// TIA Portal project "SemaforV1" (V15.1)

(* hardware
DEVICE "S71500/ET200MP station_1"  S7-1500 station
   slot 0: "Rail_0"  Rack  6ES7 590-1***0-0AA0
   slot 1: "PLC_1"  CPU 1513-1 PN  6ES7 513-1AL02-0AB0  V2.6
      slot 3: "CPU display_1"  6ES7591-1AA00-0AA0
DEVICE "HMI_1"  KTP900 Basic PN
   slot 0: "HMI_1"  KTP900 Basic PN  6AV2 123-2JB03-0AX0  15.1.0.0
   slot 1: "HMI_RT_1"  KTP900 Basic PN  6AV2 123-2JB03-0AX0  15.1.0.0
   slot 5: "HMI_1.IE_CP_1"  PROFINET Interface  15.0.1.0
      slot 1: "PROFINET Interface_1"  PROFINET Interface
         slot 1: "Port_1"  Port
*)

// ===== PLC "PLC_1"  CPU 1513-1 PN =====

VAR_GLOBAL   // PLC tag table "Default tag table"
   "Clock_Byte" AT %MB0 : Byte;
   "Clock_10Hz" AT %M0.0 : Bool;
   "Clock_5Hz" AT %M0.1 : Bool;
   "Clock_2.5Hz" AT %M0.2 : Bool;
   "Clock_2Hz" AT %M0.3 : Bool;
   "Clock_1.25Hz" AT %M0.4 : Bool;
   "Clock_1Hz" AT %M0.5 : Bool;
   "Clock_0.625Hz" AT %M0.6 : Bool;
   "Clock_0.5Hz" AT %M0.7 : Bool;
END_VAR

DATA_BLOCK "Semafor_1_variabile"   // DB1
{ S7_Optimized_Access := 'TRUE' }
VERSION : 0.1
   VAR
      "mod functionare" : UInt;
      timp_verde : Time;
      timp_galben : Time;
      timp_rosu : Time;
      verde_on : Bool;
      galben_on : Bool;
      rosu_on : Bool;
      galben_intermitent : Bool;
   END_VAR
BEGIN
END_DATA_BLOCK

DATA_BLOCK "Semafor_2_variabile"   // DB2
{ S7_Optimized_Access := 'TRUE' }
VERSION : 0.1
   VAR
      "mod functionare" : UInt;
      timp_verde : Time;
      timp_galben : Time;
      timp_rosu : Time;
      verde_on : Bool;
      galben_on : Bool;
      rosu_on : Bool;
      galben_intermitent : Bool;
   END_VAR
BEGIN
END_DATA_BLOCK

DATA_BLOCK "Semafor_3_variabile"   // DB3
{ S7_Optimized_Access := 'TRUE' }
VERSION : 0.1
   VAR
      "mod functionare" : UInt;
      timp_verde : Time;
      timp_galben : Time;
      timp_rosu : Time;
      verde_on : Bool;
      galben_on : Bool;
      rosu_on : Bool;
      galben_intermitent : Bool;
   END_VAR
BEGIN
END_DATA_BLOCK

DATA_BLOCK "Semafor2"   // DB4
{ S7_Optimized_Access := 'TRUE' }
VERSION : 0.1
// stored: InstanceOfName Semafor_fct
"Semafor_fct"
BEGIN
END_DATA_BLOCK

DATA_BLOCK "Semafor3"   // DB5
{ S7_Optimized_Access := 'TRUE' }
VERSION : 0.1
// stored: InstanceOfName Semafor_fct
"Semafor_fct"
BEGIN
END_DATA_BLOCK

DATA_BLOCK "Semafor1"   // DB6
{ S7_Optimized_Access := 'TRUE' }
VERSION : 0.1
// stored: InstanceOfName Semafor_fct
"Semafor_fct"
BEGIN
END_DATA_BLOCK

DATA_BLOCK "Semafor_4_variabile"   // DB7
{ S7_Optimized_Access := 'TRUE' }
VERSION : 0.1
   VAR
      "mod functionare" : UInt;
      timp_verde : Time;
      timp_galben : Time;
      timp_rosu : Time;
      verde_on : Bool;
      galben_on : Bool;
      rosu_on : Bool;
      galben_intermitent : Bool;
   END_VAR
BEGIN
END_DATA_BLOCK

DATA_BLOCK "Semafor4"   // DB8
{ S7_Optimized_Access := 'TRUE' }
VERSION : 0.1
// stored: InstanceOfName Semafor_fct
"Semafor_fct"
BEGIN
END_DATA_BLOCK

FUNCTION_BLOCK "Semafor_fct"   // FB1, LAD
{ S7_Optimized_Access := 'TRUE' }
VERSION : 0.1
   VAR_INPUT
      timp_verde : Time;
      timp_galben : Time;
      timp_rosu : Time;
   END_VAR
   VAR_OUTPUT
      verde_on : Bool;
      galben_on : Bool;
      rosu_on : Bool;
      galben_intermitnet : Bool;
   END_VAR
   VAR_IN_OUT
      mod_functionare : UInt;
   END_VAR
   VAR
      pornire_normal : Bool;
      reseteaza_bucla : Bool;
      porneste_verde : Bool;
      porneste_galben : Bool;
      porneste_rosu : Bool;
      timer_verde : TON_TIME;
      timer_galben : TON_TIME;
      timer_rosu : TON_TIME;
      rising_edge : Bool;
      testing : Bool;
      timp_verde_secunde : Time;
      timp_rosu_secunde : Time;
      timp_galben_secunde : Time;
   END_VAR
   VAR_TEMP   // added for the SCL form of the ladder/FBD networks
      _w1 : Bool;
   END_VAR
BEGIN

REGION Network 1: timp in secunde
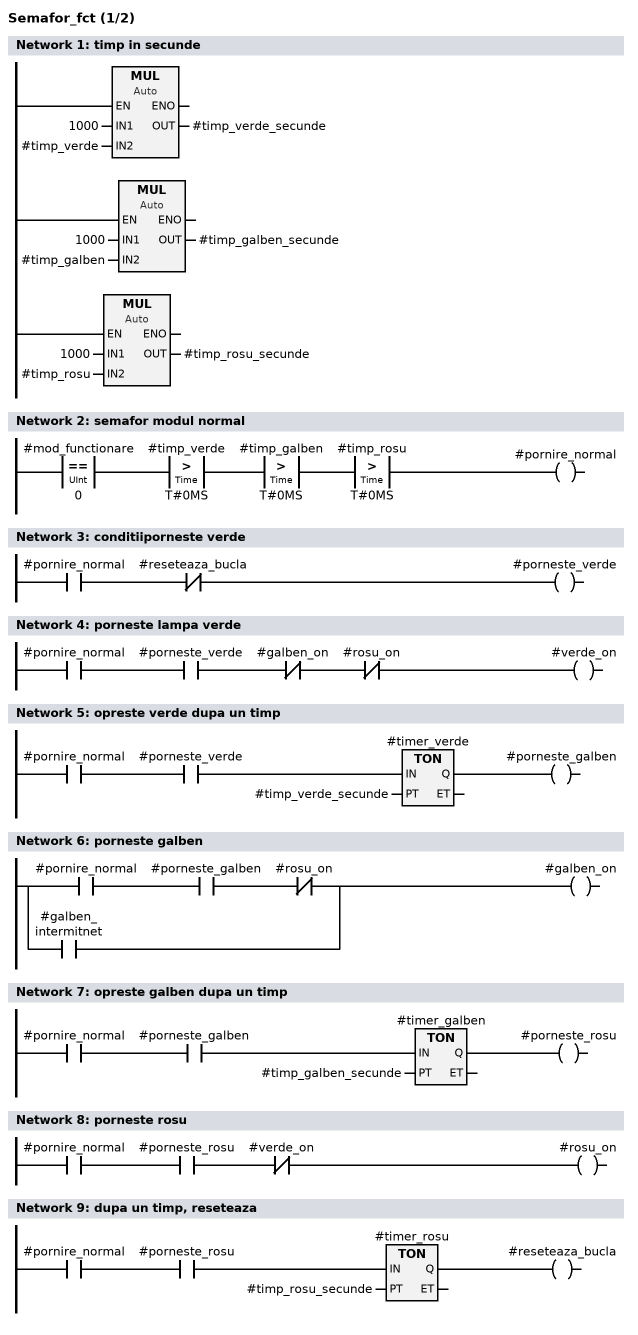
   RUNG wire#powerrail
      Mul(in1 := 1000, in2 := #timp_verde, out => #timp_verde_secunde)
   END_RUNG
   RUNG wire#powerrail
      Mul(in1 := 1000, in2 := #timp_galben, out => #timp_galben_secunde)
   END_RUNG
   RUNG wire#powerrail
      Mul(in1 := 1000, in2 := #timp_rosu, out => #timp_rosu_secunde)
   END_RUNG
   // the same network as SCL:
   #timp_verde_secunde := 1000 * #timp_verde;
   #timp_galben_secunde := 1000 * #timp_galben;
   #timp_rosu_secunde := 1000 * #timp_rosu;
END_REGION

REGION Network 2: semafor modul normal
   RUNG wire#powerrail
      { S7_Templates := "SrcType := UInt" } EQ_Contact(in1 := #mod_functionare, in2 := 0)
      { S7_Templates := "SrcType := Time" } GT_Contact(in1 := #timp_verde, in2 := T#0MS)
      { S7_Templates := "SrcType := Time" } GT_Contact(in1 := #timp_galben, in2 := T#0MS)
      { S7_Templates := "SrcType := Time" } GT_Contact(in1 := #timp_rosu, in2 := T#0MS)
      Coil( #pornire_normal )
   END_RUNG
   // the same network as SCL:
   #pornire_normal := (#mod_functionare = 0) AND (#timp_verde > T#0MS) AND (#timp_galben > T#0MS) AND (#timp_rosu > T#0MS);
END_REGION

REGION Network 3: conditiiporneste verde
   RUNG wire#powerrail
      Contact( #pornire_normal )
      I_Contact( #reseteaza_bucla )
      Coil( #porneste_verde )
   END_RUNG
   // the same network as SCL:
   #porneste_verde := #pornire_normal AND NOT #reseteaza_bucla;
END_REGION

REGION Network 4: porneste lampa verde
   RUNG wire#powerrail
      Contact( #pornire_normal )
      Contact( #porneste_verde )
      I_Contact( #galben_on )
      I_Contact( #rosu_on )
      Coil( #verde_on )
   END_RUNG
   // the same network as SCL:
   #verde_on := #pornire_normal AND #porneste_verde AND NOT #galben_on AND NOT #rosu_on;
END_REGION

REGION Network 5: opreste verde dupa un timp
   #timer_verde(IN := #pornire_normal AND #porneste_verde, PT := #timp_verde_secunde);   // TON
   #porneste_galben := #timer_verde.Q;
END_REGION

REGION Network 6: porneste galben
   RUNG wire#powerrail
      Contact( #pornire_normal )
      Contact( #porneste_galben )
      I_Contact( #rosu_on )
      wire#w1
      Coil( #galben_on )
   END_RUNG
   RUNG wire#powerrail
      Contact( #galben_intermitnet )
   END_RUNG wire#w1
   // the same network as SCL:
   #galben_on := (#pornire_normal AND #porneste_galben AND NOT #rosu_on) OR #galben_intermitnet;
END_REGION

REGION Network 7: opreste galben dupa un timp
   #timer_galben(IN := #pornire_normal AND #porneste_galben, PT := #timp_galben_secunde);   // TON
   #porneste_rosu := #timer_galben.Q;
END_REGION

REGION Network 8: porneste rosu
   RUNG wire#powerrail
      Contact( #pornire_normal )
      Contact( #porneste_rosu )
      I_Contact( #verde_on )
      Coil( #rosu_on )
   END_RUNG
   // the same network as SCL:
   #rosu_on := #pornire_normal AND #porneste_rosu AND NOT #verde_on;
END_REGION

REGION Network 9: dupa un timp, reseteaza
   #timer_rosu(IN := #pornire_normal AND #porneste_rosu, PT := #timp_rosu_secunde);   // TON
   #reseteaza_bucla := #timer_rosu.Q;
END_REGION

REGION Network 10: toggle rising edge pt SR la galben intermitent pe avarie
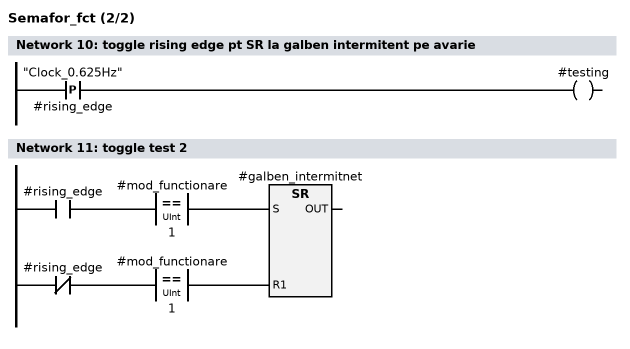
   RUNG wire#powerrail
      P_Contact(operand := "Clock_0.625Hz", bit := #rising_edge)
      Coil( #testing )
   END_RUNG
   // the same network as SCL:
   #_w1 := "Clock_0.625Hz" AND NOT #rising_edge;   // rising edge of "Clock_0.625Hz"
   #rising_edge := "Clock_0.625Hz";
   #testing := #_w1;
END_REGION

REGION Network 11: toggle test 2
   RUNG wire#powerrail
      Contact( #rising_edge )
      { S7_Templates := "SrcType := UInt" } EQ_Contact(in1 := #mod_functionare, in2 := 1)
      S_SR(operand := #galben_intermitnet, r1 := wire#w1)
   END_RUNG
   RUNG wire#powerrail
      I_Contact( #rising_edge )
      { S7_Templates := "SrcType := UInt" } EQ_Contact(in1 := #mod_functionare, in2 := 1)
   END_RUNG wire#w1
   // the same network as SCL:
   IF #rising_edge AND (#mod_functionare = 1) THEN
       #galben_intermitnet := TRUE;   // SR flip-flop
   END_IF;
   IF NOT #rising_edge AND (#mod_functionare = 1) THEN #galben_intermitnet := FALSE; END_IF;
END_REGION
END_FUNCTION_BLOCK

ORGANIZATION_BLOCK "Main"   // OB1, LAD, ProgramCycle
TITLE = "Main Program Sweep (Cycle)"
{ S7_Optimized_Access := 'TRUE' }
VERSION : 0.1
   VAR_INPUT
      Initial_Call : Bool;   // Initial call of this OB
      Remanence : Bool;   // =True, if remanent data are available
   END_VAR
   VAR_TEMP   // added for the SCL form of the ladder/FBD networks
      _w1 : Bool;
   END_VAR
BEGIN

REGION Network 1: porneste semafoarele 2 si 3 daca 1 si 4 sunt pe rosu
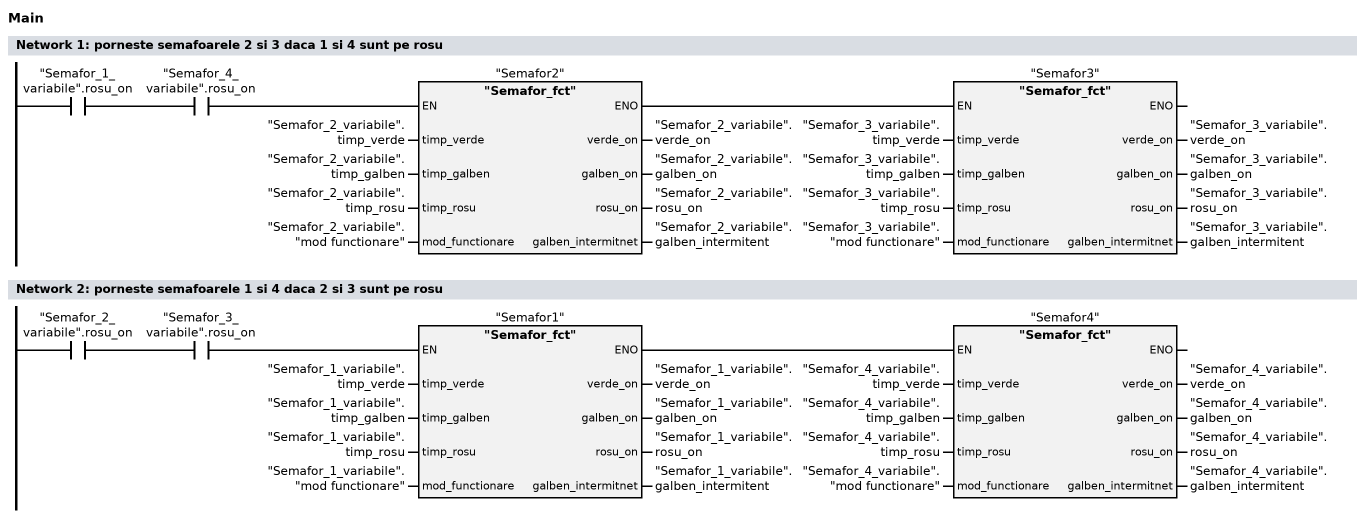
   RUNG wire#powerrail
      Contact( "Semafor_1_variabile".rosu_on )
      Contact( "Semafor_4_variabile".rosu_on )
      "Semafor2"(timp_verde := "Semafor_2_variabile".timp_verde, timp_galben := "Semafor_2_variabile".timp_galben, timp_rosu := "Semafor_2_variabile".timp_rosu, mod_functionare := "Semafor_2_variabile"."mod functionare", verde_on => "Semafor_2_variabile".verde_on, galben_on => "Semafor_2_variabile".galben_on, rosu_on => "Semafor_2_variabile".rosu_on, galben_intermitnet => "Semafor_2_variabile".galben_intermitent)
      "Semafor3"(timp_verde := "Semafor_3_variabile".timp_verde, timp_galben := "Semafor_3_variabile".timp_galben, timp_rosu := "Semafor_3_variabile".timp_rosu, mod_functionare := "Semafor_3_variabile"."mod functionare", verde_on => "Semafor_3_variabile".verde_on, galben_on => "Semafor_3_variabile".galben_on, rosu_on => "Semafor_3_variabile".rosu_on, galben_intermitnet => "Semafor_3_variabile".galben_intermitent)
   END_RUNG
   // the same network as SCL:
   "Semafor2"(EN := "Semafor_1_variabile".rosu_on AND "Semafor_4_variabile".rosu_on,   // "Semafor_fct"
              timp_verde := "Semafor_2_variabile".timp_verde,
              timp_galben := "Semafor_2_variabile".timp_galben,
              timp_rosu := "Semafor_2_variabile".timp_rosu,
              mod_functionare := "Semafor_2_variabile"."mod functionare",
              verde_on => "Semafor_2_variabile".verde_on,
              galben_on => "Semafor_2_variabile".galben_on,
              rosu_on => "Semafor_2_variabile".rosu_on,
              galben_intermitnet => "Semafor_2_variabile".galben_intermitent,
              ENO => #_w1);
   IF #_w1 THEN
       "Semafor3"(timp_verde := "Semafor_3_variabile".timp_verde,   // "Semafor_fct"
                  timp_galben := "Semafor_3_variabile".timp_galben,
                  timp_rosu := "Semafor_3_variabile".timp_rosu,
                  mod_functionare := "Semafor_3_variabile"."mod functionare",
                  verde_on => "Semafor_3_variabile".verde_on,
                  galben_on => "Semafor_3_variabile".galben_on,
                  rosu_on => "Semafor_3_variabile".rosu_on,
                  galben_intermitnet => "Semafor_3_variabile".galben_intermitent);
   END_IF;
END_REGION

REGION Network 2: porneste semafoarele 1 si 4 daca 2 si 3 sunt pe rosu
   RUNG wire#powerrail
      Contact( "Semafor_2_variabile".rosu_on )
      Contact( "Semafor_3_variabile".rosu_on )
      "Semafor1"(timp_verde := "Semafor_1_variabile".timp_verde, timp_galben := "Semafor_1_variabile".timp_galben, timp_rosu := "Semafor_1_variabile".timp_rosu, mod_functionare := "Semafor_1_variabile"."mod functionare", verde_on => "Semafor_1_variabile".verde_on, galben_on => "Semafor_1_variabile".galben_on, rosu_on => "Semafor_1_variabile".rosu_on, galben_intermitnet => "Semafor_1_variabile".galben_intermitent)
      "Semafor4"(timp_verde := "Semafor_4_variabile".timp_verde, timp_galben := "Semafor_4_variabile".timp_galben, timp_rosu := "Semafor_4_variabile".timp_rosu, mod_functionare := "Semafor_4_variabile"."mod functionare", verde_on => "Semafor_4_variabile".verde_on, galben_on => "Semafor_4_variabile".galben_on, rosu_on => "Semafor_4_variabile".rosu_on, galben_intermitnet => "Semafor_4_variabile".galben_intermitent)
   END_RUNG
   // the same network as SCL:
   "Semafor1"(EN := "Semafor_2_variabile".rosu_on AND "Semafor_3_variabile".rosu_on,   // "Semafor_fct"
              timp_verde := "Semafor_1_variabile".timp_verde,
              timp_galben := "Semafor_1_variabile".timp_galben,
              timp_rosu := "Semafor_1_variabile".timp_rosu,
              mod_functionare := "Semafor_1_variabile"."mod functionare",
              verde_on => "Semafor_1_variabile".verde_on,
              galben_on => "Semafor_1_variabile".galben_on,
              rosu_on => "Semafor_1_variabile".rosu_on,
              galben_intermitnet => "Semafor_1_variabile".galben_intermitent,
              ENO => #_w1);
   IF #_w1 THEN
       "Semafor4"(timp_verde := "Semafor_4_variabile".timp_verde,   // "Semafor_fct"
                  timp_galben := "Semafor_4_variabile".timp_galben,
                  timp_rosu := "Semafor_4_variabile".timp_rosu,
                  mod_functionare := "Semafor_4_variabile"."mod functionare",
                  verde_on => "Semafor_4_variabile".verde_on,
                  galben_on => "Semafor_4_variabile".galben_on,
                  rosu_on => "Semafor_4_variabile".rosu_on,
                  galben_intermitnet => "Semafor_4_variabile".galben_intermitent);
   END_IF;
END_REGION
END_ORGANIZATION_BLOCK

(* ===== HMI "HMI_RT_1" =====
system functions are stored by id; their names below are inferred from use
connection "HMI_Connection_1": ETHERNET, SMART_S7_1500_OMS

HMI tags "Default tag table"
   "Tag_ScreenNumber" : UInt, internal
   "Semafor_1_variabile_timp_verde" : Time = PLC Semafor_1_variabile.timp_verde, 1 s
   "Semafor_1_variabile_timp_galben" : Time = PLC Semafor_1_variabile.timp_galben, 1 s
   "Semafor_1_variabile_timp_rosu" : Time = PLC Semafor_1_variabile.timp_rosu, 1 s
   "Semafor_2_variabile_timp_verde" : Time = PLC Semafor_2_variabile.timp_verde, 1 s
   "Semafor_2_variabile_timp_galben" : Time = PLC Semafor_2_variabile.timp_galben, 1 s
   "Semafor_2_variabile_timp_rosu" : Time = PLC Semafor_2_variabile.timp_rosu, 1 s
   "Semafor_3_variabile_timp_galben" : Time = PLC Semafor_3_variabile.timp_galben, 1 s
   "Semafor_3_variabile_timp_rosu" : Time = PLC Semafor_3_variabile.timp_rosu, 1 s
   "Semafor_4_variabile_timp_verde" : Time = PLC Semafor_4_variabile.timp_verde, 1 s
   "Semafor_4_variabile_timp_galben" : Time = PLC Semafor_4_variabile.timp_galben, 1 s
   "Semafor_4_variabile_timp_rosu" : Time = PLC Semafor_4_variabile.timp_rosu, 1 s
   "Semafor_1_variabile_mod functionare" : UInt = PLC Semafor_1_variabile."mod functionare", 1 s
   "Semafor_2_variabile_mod functionare" : UInt = PLC Semafor_2_variabile."mod functionare", 1 s
   "Semafor_3_variabile_mod functionare" : UInt = PLC Semafor_3_variabile."mod functionare", 1 s
   "Semafor_4_variabile_mod functionare" : UInt = PLC Semafor_4_variabile."mod functionare", 1 s
   "Semafor_1_variabile_rosu_on" : Bool = PLC Semafor_1_variabile.rosu_on, 1 s
   "Semafor_1_variabile_galben_on" : Bool = PLC Semafor_1_variabile.galben_on, 1 s
   "Semafor_1_variabile_verde_on" : Bool = PLC Semafor_1_variabile.verde_on, 1 s
   "Semafor_2_variabile_rosu_on" : Bool = PLC Semafor_2_variabile.rosu_on, 1 s
   "Semafor_2_variabile_galben_on" : Bool = PLC Semafor_2_variabile.galben_on, 1 s
   "Semafor_2_variabile_verde_on" : Bool = PLC Semafor_2_variabile.verde_on, 1 s
   "Semafor_3_variabile_rosu_on" : Bool = PLC Semafor_3_variabile.rosu_on, 1 s
   "Semafor_3_variabile_galben_on" : Bool = PLC Semafor_3_variabile.galben_on, 1 s
   "Semafor_3_variabile_verde_on" : Bool = PLC Semafor_3_variabile.verde_on, 1 s
   "Semafor_4_variabile_verde_on" : Bool = PLC Semafor_4_variabile.verde_on, 1 s
   "Semafor_4_variabile_galben_on" : Bool = PLC Semafor_4_variabile.galben_on, 1 s
   "Semafor_4_variabile_rosu_on" : Bool = PLC Semafor_4_variabile.rosu_on, 1 s

Template "Template_1" 800x480
   Button "Exit" at 722,440 size 55x39; TextOff 'Exit'; PictureOff "ExitRuntime_KTP900_Basic_PN_TR"; PictureOn "ExitRuntime_KTP900_Basic_PN_TR"
      on Release: StopRuntime(0)
   Button "Template_Button" at 622,440 size 55x39; TextOff 'Text'
   Button "Template_Button_1" at 522,440 size 55x39; TextOff 'Text'
   Button "Template_Button_2" at 422,440 size 55x39; TextOff 'Text'
   Button "Template_Button_3" at 322,440 size 55x39; TextOff 'Text'
   Button "Template_Button_4" at 222,440 size 55x39; TextOff 'Text'
   Button "Alarms" at 122,440 size 55x39; TextOff 'Alarms'; PictureOff "AlarmDisplay_KTP900_Basic_PN_TR"; PictureOn "AlarmDisplay_KTP900_Basic_PN_TR"
   Button "Start screen" at 22,440 size 55x39; TextOff 'Start screen'; PictureOff "NavigateHome_KTP900_Basic_PN_TR"; PictureOn "NavigateHome_KTP900_Basic_PN_TR"
      on Release: ActivateScreen("Simulare", 0)
   SymbolicIOField "Symbolic_IO_Field_Screen" at 73,7 size 620x26; TextOff '0'; TextOn '1'; TextList "TextList_ScreenNames"
      ProcessValue <- "Tag_ScreenNumber"
      on Change: ActivateScreenByNumber("Tag_ScreenNumber", 0)
   DateTimeField "HmiScreenItemData" at 695,20 size 105x20
   DateTimeField "HmiScreenItemData_1" at 695,0 size 105x20
   GraphicView "Logo" at 0,0 size 71x40; Picture "Logo of HMI_1"

screen "Simulare" 800x480, template "Template_1"
   on GenerateScreen: SetTag("Tag_ScreenNumber", 1)
   TextField "Text field_1" at 462,283 size 13x20; Text '1'
   TextField "Text field_2" at 461,173 size 13x20; Text '2'
   TextField "Text field_3" at 307,288 size 13x20; Text '3'
   TextField "Text field_4" at 308,173 size 13x20; Text '4'
   TextField "Text field_5" at 496,314 size 19x25; Text '^'
   TextField "Text field_6" at 499,328 size 12x20; Text '|'
   TextField "Text field_7" at 489,173 size 22x20; Text '<-'
   TextField "Text field_8" at 299,328 size 22x20; Text '->'
   Circle "Circle_1" at 482,286 size 7x7
      Appearance <- "Semafor_1_variabile_rosu_on"
   Circle "Circle_2" at 482,294 size 7x7
      Appearance <- "Semafor_1_variabile_galben_on"
   Circle "Circle_3" at 482,303 size 7x7
      Appearance <- "Semafor_1_variabile_verde_on"
   Circle "Circle_4" at 482,132 size 7x7
      Appearance <- "Semafor_2_variabile_rosu_on"
   Circle "Circle_5" at 482,140 size 7x7
      Appearance <- "Semafor_2_variabile_galben_on"
   Circle "Circle_6" at 482,149 size 7x7
      Appearance <- "Semafor_2_variabile_verde_on"
   Circle "Circle_7" at 290,132 size 7x7
      Appearance <- "Semafor_4_variabile_rosu_on"
   Circle "Circle_8" at 290,140 size 7x7
      Appearance <- "Semafor_4_variabile_galben_on"
   Circle "Circle_9" at 290,149 size 7x7
      Appearance <- "Semafor_4_variabile_verde_on"
   Circle "Circle_10" at 290,289 size 7x7
      Appearance <- "Semafor_3_variabile_rosu_on"
   Circle "Circle_11" at 290,297 size 7x7
      Appearance <- "Semafor_3_variabile_galben_on"
   Circle "Circle_12" at 290,306 size 7x7
      Appearance <- "Semafor_3_variabile_verde_on"

screen "Comenzi" 800x480
   IOField "I/O field_1" at 26,205 size 96x32; FormatPattern 999; Unit s
      ProcessValue <- "Semafor_1_variabile_timp_verde"
   TextField "Text field_1" at 26,175 size 82x20; Text 'Timer verde'
   IOField "I/O field_2" at 26,278 size 96x32; FormatPattern 999; Unit s
      ProcessValue <- "Semafor_1_variabile_timp_galben"
   TextField "Text field_2" at 26,248 size 87x20; Text 'Timer galben'
   IOField "I/O field_3" at 26,352 size 96x32; FormatPattern 999; Unit s
      ProcessValue <- "Semafor_1_variabile_timp_rosu"
   TextField "Text field_3" at 26,321 size 73x20; Text 'Timer rosu'
   IOField "I/O field_4" at 176,205 size 96x32; FormatPattern 999; Unit s
      ProcessValue <- "Semafor_2_variabile_timp_verde"
   TextField "Text field_4" at 176,175 size 82x20; Text 'Timer verde'
   IOField "I/O field_5" at 176,278 size 96x32; FormatPattern 999; Unit s
      ProcessValue <- "Semafor_2_variabile_timp_galben"
   TextField "Text field_5" at 176,248 size 87x20; Text 'Timer galben'
   IOField "I/O field_6" at 176,352 size 96x32; FormatPattern 999; Unit s
      ProcessValue <- "Semafor_2_variabile_timp_rosu"
   TextField "Text field_6" at 176,321 size 73x20; Text 'Timer rosu'
   IOField "I/O field_7" at 326,205 size 96x32; FormatPattern 999; Unit s
      ProcessValue <- "Semafor_3_variabile_timp_galben"
   TextField "Text field_7" at 326,175 size 82x20; Text 'Timer verde'
   IOField "I/O field_8" at 326,278 size 96x32; FormatPattern 999; Unit s
      ProcessValue <- "Semafor_3_variabile_timp_galben"
   TextField "Text field_8" at 326,248 size 87x20; Text 'Timer galben'
   IOField "I/O field_9" at 326,352 size 96x32; FormatPattern 999; Unit s
      ProcessValue <- "Semafor_3_variabile_timp_rosu"
   TextField "Text field_9" at 326,321 size 73x20; Text 'Timer rosu'
   IOField "I/O field_10" at 476,205 size 96x32; FormatPattern 999; Unit s
      ProcessValue <- "Semafor_4_variabile_timp_verde"
   TextField "Text field_10" at 476,175 size 82x20; Text 'Timer verde'
   IOField "I/O field_11" at 476,278 size 96x32; FormatPattern 999; Unit s
      ProcessValue <- "Semafor_4_variabile_timp_galben"
   TextField "Text field_11" at 476,248 size 87x20; Text 'Timer galben'
   IOField "I/O field_12" at 476,352 size 96x32; FormatPattern 999; Unit s
      ProcessValue <- "Semafor_4_variabile_timp_rosu"
   TextField "Text field_12" at 476,321 size 73x20; Text 'Timer rosu'
   TextField "Text field_13" at 47,133 size 71x20; Text 'Semafor 1'
   TextField "Text field_14" at 198,133 size 71x20; Text 'Semafor 2'
   TextField "Text field_15" at 347,133 size 71x20; Text 'Semafor 3'
   TextField "Text field_16" at 491,133 size 71x20; Text 'Semafor 4'
   Button "Button_1" at 35,23 size 96x32; TextOff 'Mod Normal'
      on Click: SetTag("Semafor_1_variabile_mod functionare", 0)
   Button "Button_2" at 35,75 size 96x32; TextOff 'Mod Avarie'
      on Click: SetTag("Semafor_1_variabile_mod functionare", 1)
   Button "Button_3" at 185,25 size 96x32; TextOff 'Mod Normal'
      on Click: SetTag("Semafor_2_variabile_mod functionare", 0)
   Button "Button_4" at 185,77 size 96x32; TextOff 'Mod Avarie'
      on Click: SetTag("Semafor_2_variabile_mod functionare", 1)
   Button "Button_5" at 334,27 size 96x32; TextOff 'Mod Normal'
      on Click: SetTag("Semafor_3_variabile_mod functionare", 0)
   Button "Button_6" at 334,79 size 96x32; TextOff 'Mod Avarie'
      on Click: SetTag("Semafor_3_variabile_mod functionare", 1)
   Button "Button_7" at 484,29 size 96x32; TextOff 'Mod Normal'
      on Click: SetTag("Semafor_4_variabile_mod functionare", 0)
   Button "Button_8" at 484,81 size 96x32; TextOff 'Mod Avarie'
      on Click: SetTag("Semafor_4_variabile_mod functionare", 1)
*)